{attribute 'linkalways'} 
{attribute 'no_explicit_call' := 'This FB is a CLASS and must be accessed using methods or properties'}
{attribute 'enable_dynamic_creation'}
FUNCTION_BLOCK Node_F_VN_DrawOrientation EXTENDS VisionNode
VAR
    stOrientation : _TcVnRotatedRectangle;
    ipDestImage : _ITcVnImage;
    aColorMainAxis : _TcVnVector4_LREAL;
    nThickness : _DINT(1);
    hrPrev : _HRESULT(S_OK);
	hresult : _HRESULT(S_OK);
END_VAR

METHOD PUBLIC  Clone : I_Node
VAR
	pNode : POINTER TO Node_F_VN_DrawOrientation;
END_VAR
pNode := __NEW(Node_F_VN_DrawOrientation);
Clone := pNode^;
END_METHOD

METHOD FB_init : BOOL
VAR_INPUT
	bInitRetains : BOOL; // if TRUE, the retain variables are initialized (warm start / cold start)
	bInCopyCode : BOOL;  // if TRUE, the instance afterwards gets moved into the copy code (online change)
END_VAR
AddInput('stOrientation', stOrientation);
AddInput('ipDestImage', ipDestImage);
AddInput('aColorMainAxis', aColorMainAxis);
AddParameter('nThickness', nThickness);
AddInput('hrPrev', hrPrev);
AddOutput('ipDestImage', ipDestImage);
AddOutput('hresult',hresult);
END_METHOD

METHOD PROTECTED OnExecute
hresult.Value := F_VN_DrawOrientation(
    stOrientation := stOrientation.Value,
	ipDestImage := ipDestImage.Value,
    aColorMainAxis := aColorMainAxis.Value,
    nThickness := nThickness.Value,
	hrPrev:= hrPrev.Value);
END_METHOD

METHOD PUBLIC PreExecutionCheck
VAR_INPUT
	Check : I_PreExecutionChecks;
END_VAR
Check.IsTrue(ipDestImage.IsValid, 'ipDestImage must contain an image');
Check.IsTrue(nThickness.Value >= 1, 'nThickness must be greater than or equal to 1');
END_METHOD

END_FUNCTION_BLOCK

(* stored: Version 1.1.0.1, ProductVersion 3.1.4024.15
   POU Node_F_VN_DrawOrientation: Id {403b8853-07e2-07ba-1e55-c0ed83d9904a}, SpecialFunc None
   Folder Constructor: Id {bee3675a-2ce6-0a95-18b0-4c12ff8ff211}
   Method Clone: Id {babf7a86-e09d-064b-399b-1e9e59e364bf}
   Method FB_init: Id {43d3ac1d-3f2f-0efe-0037-b6b96839e33c}
   Method OnExecute: Id {c23b8a57-b4c2-07fe-160e-1ad0ef47cea1}
   Method PreExecutionCheck: Id {76d159c7-10c8-0be0-1d7e-9816aba2850f} *)
